FUNCTION_BLOCK Setup (* Basic Function Block Type *)
  (* Standard: 61499-2 *)
  (* Version 0.0, 21/06/2022, Lernfabrik, WBK hackaton, Template *)
  PACKAGE Main;
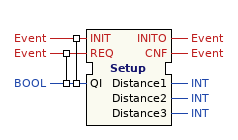
  EVENT_INPUT
    INIT WITH QI; (* Initialization Request *)
    REQ WITH QI; (* Normal Execution Request *)
  END_EVENT
  EVENT_OUTPUT
    INITO; (* Initialization Confirm *)
    CNF; (* Execution Confirmation *)
  END_EVENT
  VAR_INPUT
    QI : BOOL; (* Input event qualifier *)
  END_VAR
  VAR_OUTPUT
    Distance1 : INT;
    Distance2 : INT;
    Distance3 : INT;
  END_VAR
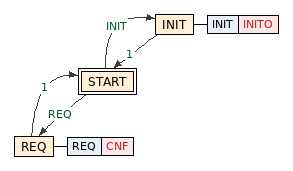
  EC_STATES
    START; (* Initial State *)
    INIT : INIT -> INITO; (* Initialization *)
    REQ : REQ -> CNF; (* Normal execution *)
  END_STATES
  EC_TRANSITIONS
    START TO INIT := INIT;
    INIT TO START := 1;
    START TO REQ := REQ;
    REQ TO START := 1;
  END_TRANSITIONS
  ALGORITHM INIT IN ST: (* Initialization algorithm *)
;
  END_ALGORITHM
  ALGORITHM REQ IN ST: (* Normally executed algorithm *)
;
  END_ALGORITHM
END_FUNCTION_BLOCK
